// TIA Portal project "Hardware Configuration 9" (V15.1)

(* hardware
DEVICE "S71500/ET200MP station_1"  S7-1500 station
   slot 0: "Rail_0"  Rack  6ES7 590-1***0-0AA0
   slot 0: "PM 190W 120/230VAC"  PM 190W 120/230VAC  6EP1333-4BA00
   slot 1: "PLC_1"  CPU 1516-3 PN/DP  6ES7 516-3AN01-0AB0  V2.6
      slot 3: "CPU display_1"  6ES7591-1BA00-0AA0
   slot 2: "DQ 32x24VDC/0.5A HF_1"  DQ 32x24VDC/0.5A HF  6ES7 522-1BL01-0AB0  V1.1
   slot 3: "DI 32x24VDC HF_1"  DI 32x24VDC HF  6ES7 521-1BL00-0AB0  V2.1
   slot 4: "AQ 4xU/I ST_1"  AQ 4xU/I ST  6ES7 532-5HD00-0AB0  V2.2
   slot 5: "AI 8xU/I/RTD/TC ST_1"  AI 8xU/I/RTD/TC ST  6ES7 531-7KF00-0AB0  V2.2
*)

// ===== PLC "PLC_1"  CPU 1516-3 PN/DP =====

VAR_GLOBAL   // PLC tag table "Full_Tag_Table"
   "Panel Emergency Stop" AT %I2.7 : Bool;
   "Start switch" AT %I0.2 : Bool;
   "Stop switch" AT %I0.3 : Bool;
   "Sort area IR" AT %I0.4 : Bool;
   "Sort Area Inductive" AT %I0.5 : Bool;
   "Sort Solenoid Sensor" AT %I0.6 : Bool;
   "Assembly Chute IR" AT %I0.7 : Bool;
   "Assembly Area Through Beam" AT %I1.1 : Bool;
   "Assembly Area Capacitor" AT %I1.2 : Bool;
   "Assembly Area Inductive" AT %I1.3 : Bool;
   "Reject Area IR" AT %I1.4 : Bool;
   "Reject Solenoid Sensor" AT %I1.5 : Bool;
   "Oven Through Beam" AT %I1.6 : Bool;
   "Loading Area Inductive" AT %I1.7 : Bool;
   "Chain Conveyor" AT %Q0.0 : Bool;
   "Sort Solenoid" AT %Q0.1 : Bool;
   "Reject Solenoid" AT %Q0.2 : Bool;
   "Rotary Solenoid" AT %Q0.3 : Bool;
   "Belt Conveyor Direction" AT %Q0.4 : Bool;
   "System Run_Green Lamp" AT %Q3.0 : Bool;
   "Sysyem Stop_Red Lamp" AT %Q3.2 : Bool;
   "Emergency stop" AT %I1.0 : Bool;
   "Ring Queue counter Full" AT %M4.0 : Bool;
   "Sort Solenoid error" AT %M4.3 : Bool;
   "Counter value" AT %MW0 : Int;
   "Reject Solenoid Error" AT %M4.7 : Bool;
   "HMI_Start" AT %M4.1 : Bool;
   "HMI_Stop" AT %M4.2 : Bool;
   "Counter Reset" AT %M4.4 : Bool;
   "DO_card" AT %QD0 : DWord;
   "DI_card" AT %ID0 : DWord;
END_VAR

DATA_BLOCK "Conveyors_AUTOMATIC_DB"   // DB1
{ S7_Optimized_Access := 'TRUE' }
VERSION : 0.1
// stored: InstanceOfName Conveyors_AUTOMATIC
"Conveyors_AUTOMATIC"
BEGIN
END_DATA_BLOCK

DATA_BLOCK "Sort Solenoid active_DB"   // DB2
{ S7_Optimized_Access := 'TRUE' }
VERSION : 0.1
// stored: InstanceOfName Sort Solenoid active
"Sort Solenoid active"
BEGIN
END_DATA_BLOCK

DATA_BLOCK "Sort Solenoid active_DB_1"   // DB3
{ S7_Optimized_Access := 'TRUE' }
VERSION : 0.1
// stored: InstanceOfName Sort Solenoid active
"Sort Solenoid active"
BEGIN
END_DATA_BLOCK

DATA_BLOCK "Solenoid Error_DB"   // DB4
{ S7_Optimized_Access := 'TRUE' }
VERSION : 0.1
// stored: InstanceOfName Solenoid Error
"Solenoid Error"
BEGIN
END_DATA_BLOCK

DATA_BLOCK "Counting_DB"   // DB5
{ S7_Optimized_Access := 'TRUE' }
VERSION : 0.1
// stored: InstanceOfName Counting
"Counting"
BEGIN
END_DATA_BLOCK

DATA_BLOCK "Rotary Solenoid1_DB"   // DB6
{ S7_Optimized_Access := 'TRUE' }
VERSION : 0.1
// stored: InstanceOfName Rotary Solenoid1
"Rotary Solenoid1"
BEGIN
END_DATA_BLOCK

FUNCTION_BLOCK "Conveyors_AUTOMATIC"   // FB1, LAD
TITLE = Conveyors Automatic
{ S7_Optimized_Access := 'TRUE' }
VERSION : 0.1
   VAR_INPUT
      "Start Switch" : Bool;
      "Stop Switch" : Bool;
      "Emergency Stop" : Bool;
      "Sort Solenoid Error" : Bool;
      "Panel Emergency Stop" : Bool;
   END_VAR
   VAR_OUTPUT
      "Chain Conveyor" : Bool;
      "Belt Conveyor" : Bool;
      "System Enable_OK" : Bool;
      "System Enable_not_OK" : Bool;
   END_VAR
   VAR
      Memory_Automatic_Start_Stop : Bool;
   END_VAR
BEGIN

REGION Network 1: System Enable_OK and Conveyor Run
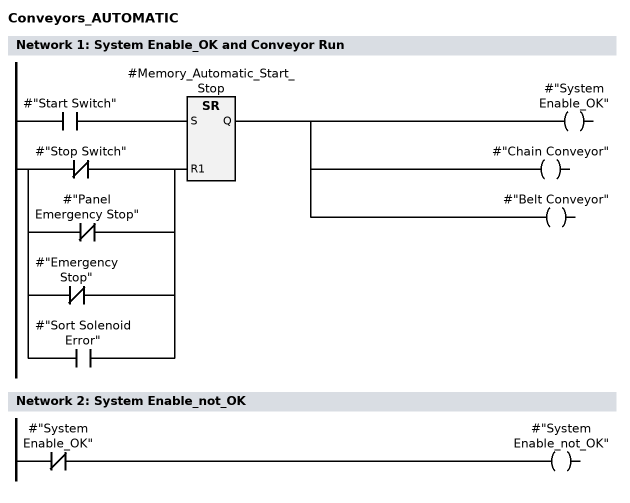
   RUNG wire#powerrail
      Contact( #"Start Switch" )
      S_SR(operand := #Memory_Automatic_Start_Stop, r1 := wire#w1)
      wire#w2
      Coil( #"System Enable_OK" )
   END_RUNG
   RUNG wire#powerrail
      I_Contact( #"Stop Switch" )
   END_RUNG wire#w1
   RUNG wire#powerrail
      I_Contact( #"Panel Emergency Stop" )
   END_RUNG wire#w1
   RUNG wire#powerrail
      I_Contact( #"Emergency Stop" )
   END_RUNG wire#w1
   RUNG wire#powerrail
      Contact( #"Sort Solenoid Error" )
   END_RUNG wire#w1
   RUNG wire#w2
      Coil( #"Chain Conveyor" )
   END_RUNG
   RUNG wire#w2
      Coil( #"Belt Conveyor" )
   END_RUNG
   // the same network as SCL:
   IF #"Start Switch" THEN
       #Memory_Automatic_Start_Stop := TRUE;   // SR flip-flop
   END_IF;
   IF NOT #"Stop Switch" OR NOT #"Panel Emergency Stop" OR NOT #"Emergency Stop" OR #"Sort Solenoid Error" THEN
       #Memory_Automatic_Start_Stop := FALSE;
   END_IF;
   #"System Enable_OK" := #Memory_Automatic_Start_Stop;
   #"Chain Conveyor" := #Memory_Automatic_Start_Stop;
   #"Belt Conveyor" := #Memory_Automatic_Start_Stop;
END_REGION

REGION Network 2: System Enable_not_OK
   RUNG wire#powerrail
      I_Contact( #"System Enable_OK" )
      Coil( #"System Enable_not_OK" )
   END_RUNG
   // the same network as SCL:
   #"System Enable_not_OK" := NOT #"System Enable_OK";
END_REGION
END_FUNCTION_BLOCK

FUNCTION_BLOCK "Sort Solenoid active"   // FB2, LAD
TITLE = Sort Solenoid active
{ S7_Optimized_Access := 'TRUE' }
VERSION : 0.1
   VAR_INPUT
      "Sort Area IR" : Bool;
      "Sort Area Inductive" : Bool;
      "Ring Queue counter full" : Bool;
   END_VAR
   VAR_OUTPUT
      "Sort Solenoid" : Bool;
   END_VAR
   VAR
      "Component Pass Delay" : Bool;
      "SR_Sort solenoid on Timer" : Bool;
      "SR_Component pass Delay" : Bool;
      IEC_Timer_0_Instance : TON_TIME;
      IEC_Timer_0_Instance_1 : TON_TIME;
   END_VAR
BEGIN

REGION Network 1: Sort Solenoid activate in case of plastic ring presence
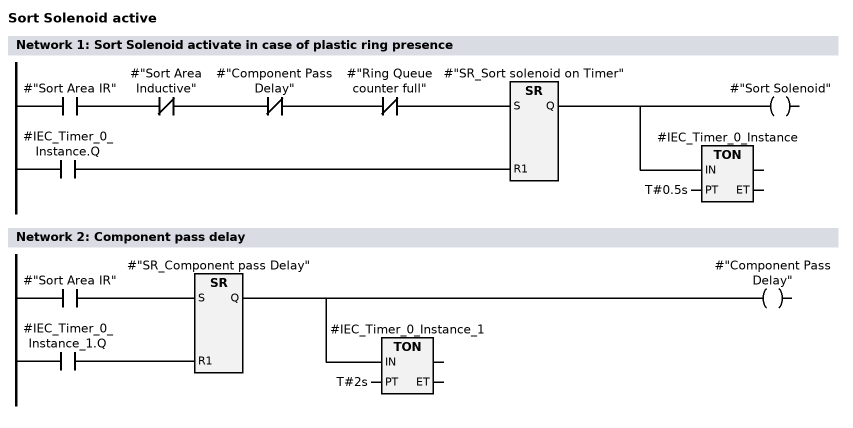
   IF #"Sort Area IR" AND NOT #"Sort Area Inductive" AND NOT #"Component Pass Delay" AND NOT #"Ring Queue counter full" THEN
       #"SR_Sort solenoid on Timer" := TRUE;   // SR flip-flop
   END_IF;
   IF #IEC_Timer_0_Instance.Q THEN #"SR_Sort solenoid on Timer" := FALSE; END_IF;
   #"Sort Solenoid" := #"SR_Sort solenoid on Timer";
   #IEC_Timer_0_Instance(IN := #"SR_Sort solenoid on Timer", PT := T#0.5s);   // TON
END_REGION

REGION Network 2: Component pass delay
   IF #"Sort Area IR" THEN
       #"SR_Component pass Delay" := TRUE;   // SR flip-flop
   END_IF;
   IF #IEC_Timer_0_Instance_1.Q THEN #"SR_Component pass Delay" := FALSE; END_IF;
   #"Component Pass Delay" := #"SR_Component pass Delay";
   #IEC_Timer_0_Instance_1(IN := #"SR_Component pass Delay", PT := T#2s);   // TON
END_REGION
END_FUNCTION_BLOCK

FUNCTION_BLOCK "Solenoid Error"   // FB3, LAD
TITLE = Solenoid error
{ S7_Optimized_Access := 'TRUE' }
VERSION : 0.1
   VAR_INPUT
      "Solenoid on" : Bool;
      "Solenoid sensor" : Bool;
   END_VAR
   VAR_OUTPUT
      "Solenoid error" : Bool;
   END_VAR
   VAR
      "Hold off delay" : Bool;
      IEC_Timer_0_Instance : TON_TIME;
   END_VAR
BEGIN

REGION Network 1: Solenoid error
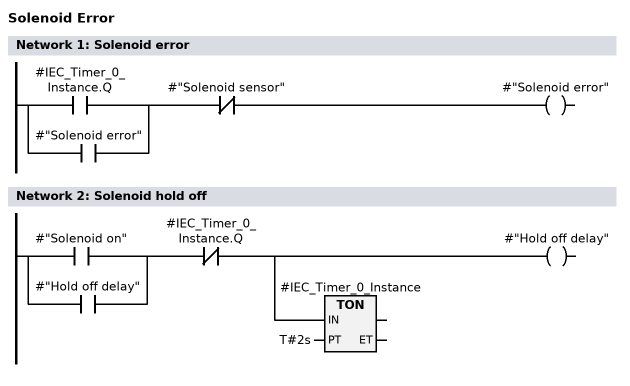
   RUNG wire#powerrail
      Contact( #IEC_Timer_0_Instance.Q )
      wire#w1
      I_Contact( #"Solenoid sensor" )
      Coil( #"Solenoid error" )
   END_RUNG
   RUNG wire#powerrail
      Contact( #"Solenoid error" )
   END_RUNG wire#w1
   // the same network as SCL:
   #"Solenoid error" := (#IEC_Timer_0_Instance.Q OR #"Solenoid error") AND NOT #"Solenoid sensor";
END_REGION

REGION Network 2: Solenoid hold off
   #"Hold off delay" := (#"Solenoid on" OR #"Hold off delay") AND NOT #IEC_Timer_0_Instance.Q;
   #IEC_Timer_0_Instance(IN := #"Hold off delay", PT := T#2s);   // TON
END_REGION
END_FUNCTION_BLOCK

FUNCTION_BLOCK "Counting"   // FB4, LAD
{ S7_Optimized_Access := 'TRUE' }
VERSION : 0.1
   VAR_INPUT
      "Sort Solenoid" : Bool;
      "Rotary Solenoid" : Bool;
      "Reset counter" : Bool;
      "Stop switch" : Bool;
   END_VAR
   VAR_OUTPUT
      "Counter value" : Int;
      "Ring Queue counter full" : Bool;
   END_VAR
   VAR RETAIN
      IEC_Counter_0_Instance : CTUD_INT;
   END_VAR
BEGIN

REGION Network 1
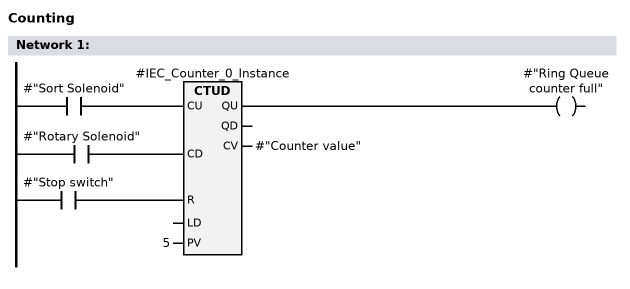
   #IEC_Counter_0_Instance(CU := #"Sort Solenoid",   // CTUD
                           CD := #"Rotary Solenoid",
                           R := #"Stop switch",
                           PV := 5,
                           CV => #"Counter value");
   #"Ring Queue counter full" := #IEC_Counter_0_Instance.QU;
END_REGION
END_FUNCTION_BLOCK

FUNCTION_BLOCK "Rotary Solenoid1"   // FB5, LAD
{ S7_Optimized_Access := 'TRUE' }
VERSION : 0.1
   VAR_INPUT
      "Assembly chute IR" : Bool;
      "Counter value" : Int;
   END_VAR
   VAR_OUTPUT
      "Rotary Solenoid" : Bool;
   END_VAR
   VAR
      "Rotary Solenoid on Timer" : Bool;
      IEC_Timer_0_Instance : TON_TIME;
   END_VAR
BEGIN

REGION Network 1: Rotary Solenoid
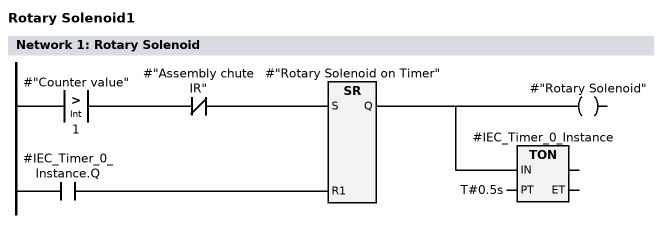
   IF (#"Counter value" > 1) AND NOT #"Assembly chute IR" THEN
       #"Rotary Solenoid on Timer" := TRUE;   // SR flip-flop
   END_IF;
   IF #IEC_Timer_0_Instance.Q THEN #"Rotary Solenoid on Timer" := FALSE; END_IF;
   #"Rotary Solenoid" := #"Rotary Solenoid on Timer";
   #IEC_Timer_0_Instance(IN := #"Rotary Solenoid on Timer", PT := T#0.5s);   // TON
END_REGION
END_FUNCTION_BLOCK

ORGANIZATION_BLOCK "Main"   // OB1, LAD, ProgramCycle
TITLE = "Main Program Sweep (Cycle)"
{ S7_Optimized_Access := 'TRUE' }
VERSION : 0.1
   VAR_INPUT
      Initial_Call : Bool;   // Initial call of this OB
      Remanence : Bool;   // =True, if remanent data are available
   END_VAR
BEGIN

REGION Network 1: System Run OK and conveyors start
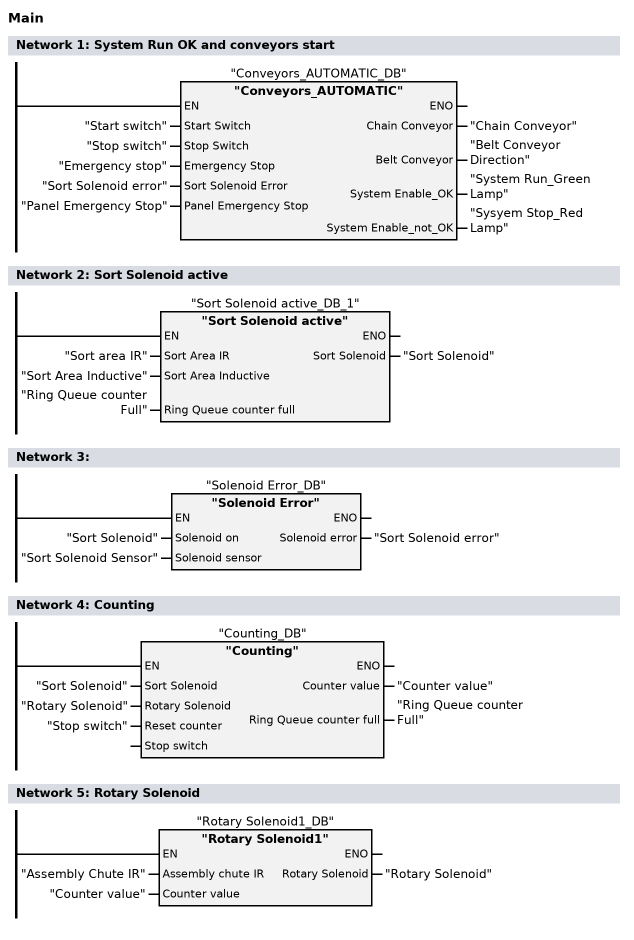
   RUNG wire#powerrail
      "Conveyors_AUTOMATIC_DB"("Start Switch" := "Start switch", "Stop Switch" := "Stop switch", "Emergency Stop" := "Emergency stop", "Sort Solenoid Error" := "Sort Solenoid error", "Panel Emergency Stop" := "Panel Emergency Stop", "Chain Conveyor" => "Chain Conveyor", "Belt Conveyor" => "Belt Conveyor Direction", "System Enable_OK" => "System Run_Green Lamp", "System Enable_not_OK" => "Sysyem Stop_Red Lamp")
   END_RUNG
   // the same network as SCL:
   "Conveyors_AUTOMATIC_DB"("Start Switch" := "Start switch",   // "Conveyors_AUTOMATIC"
                           "Stop Switch" := "Stop switch",
                           "Emergency Stop" := "Emergency stop",
                           "Sort Solenoid Error" := "Sort Solenoid error",
                           "Panel Emergency Stop" := "Panel Emergency Stop",
                           "Chain Conveyor" => "Chain Conveyor",
                           "Belt Conveyor" => "Belt Conveyor Direction",
                           "System Enable_OK" => "System Run_Green Lamp",
                           "System Enable_not_OK" => "Sysyem Stop_Red Lamp");
END_REGION

REGION Network 2: Sort Solenoid active
   RUNG wire#powerrail
      "Sort Solenoid active_DB_1"("Sort Area IR" := "Sort area IR", "Sort Area Inductive" := "Sort Area Inductive", "Ring Queue counter full" := "Ring Queue counter Full", "Sort Solenoid" => "Sort Solenoid")
   END_RUNG
   // the same network as SCL:
   "Sort Solenoid active_DB_1"("Sort Area IR" := "Sort area IR",   // "Sort Solenoid active"
                           "Sort Area Inductive" := "Sort Area Inductive",
                           "Ring Queue counter full" := "Ring Queue counter Full",
                           "Sort Solenoid" => "Sort Solenoid");
END_REGION

REGION Network 3
   RUNG wire#powerrail
      "Solenoid Error_DB"("Solenoid on" := "Sort Solenoid", "Solenoid sensor" := "Sort Solenoid Sensor", "Solenoid error" => "Sort Solenoid error")
   END_RUNG
   // the same network as SCL:
   "Solenoid Error_DB"("Solenoid on" := "Sort Solenoid",   // "Solenoid Error"
                       "Solenoid sensor" := "Sort Solenoid Sensor",
                       "Solenoid error" => "Sort Solenoid error");
END_REGION

REGION Network 4: Counting
   RUNG wire#powerrail
      "Counting_DB"("Sort Solenoid" := "Sort Solenoid", "Rotary Solenoid" := "Rotary Solenoid", "Reset counter" := "Stop switch", "Stop switch" :=, "Counter value" => "Counter value", "Ring Queue counter full" => "Ring Queue counter Full")
   END_RUNG
   // the same network as SCL:
   "Counting_DB"("Sort Solenoid" := "Sort Solenoid",   // "Counting"
                 "Rotary Solenoid" := "Rotary Solenoid",
                 "Reset counter" := "Stop switch",
                 "Counter value" => "Counter value",
                 "Ring Queue counter full" => "Ring Queue counter Full");
END_REGION

REGION Network 5: Rotary Solenoid
   RUNG wire#powerrail
      "Rotary Solenoid1_DB"("Assembly chute IR" := "Assembly Chute IR", "Counter value" := "Counter value", "Rotary Solenoid" => "Rotary Solenoid")
   END_RUNG
   // the same network as SCL:
   "Rotary Solenoid1_DB"("Assembly chute IR" := "Assembly Chute IR",   // "Rotary Solenoid1"
                         "Counter value" := "Counter value",
                         "Rotary Solenoid" => "Rotary Solenoid");
END_REGION
END_ORGANIZATION_BLOCK